
FUNCTION CB_word_to_byte : BYTE

TITLE = ' Convert a word into a byte '
VERSION : '1.0'
AUTHOR  : CB
NAME    : DworToBy
FAMILY  : TNI

VAR_INPUT
    IN : WORD;
END_VAR

VAR_TEMP

END_VAR

BEGIN

CB_word_to_byte := WORD_TO_BYTE(IN);

END_FUNCTION
